// TwinCAT 3 PLC project Test
// ProgramVersion: 3.1.4026.20
// libraries:
//   AUT_Utilities, * (AU-tomation)
//   Tc2_Standard, * (Beckhoff Automation GmbH)
//   Tc2_System, * (Beckhoff Automation GmbH)
//   Tc2_Utilities, * (Beckhoff Automation GmbH)
//   TcUnit, * (www.tcunit.org)
// project tree:
//   / PlcTask.TcTTO
//   POUs/ PRG_TEST.TcPOU, StringBuilder_Test.TcPOU
// real-time tasks:
//   TASK PlcTask: cycle T#10ms, priority 20, ADS port 350

CONFIGURATION Test
    RESOURCE PLC ON TwinCAT3
        TASK PlcTask(INTERVAL := T#10ms, PRIORITY := 20);
        PROGRAM PRG_TEST WITH PlcTask : PRG_TEST;
    END_RESOURCE
END_CONFIGURATION

// ---- POUs/PRG_TEST.TcPOU
{attribute 'no-analysis'}       // Disable SA for entire POU
PROGRAM PRG_TEST
VAR
    {attribute 'analysis' := '-33'}      // Disable SA0033: Unused variable
    _StringBuilder_Test : StringBuilder_Test;
END_VAR

//TcUnit.RUN();
TcUnit.RUN_IN_SEQUENCE();

END_PROGRAM

// ---- POUs/StringBuilder_Test.TcPOU
{attribute 'no-analysis'}       // Disable SA for entire POU
FUNCTION_BLOCK StringBuilder_Test EXTENDS TcUnit.FB_TestSuite

ToStringWithoutAppendEqualsEmptyString();
AppendABCTo123EqualsABC123();
AppendWithFormat();
LeftOfABC123With3EqualsABC();
RightOfABC123With3Equals123();
InsertXYZAt3IntoABC123EqualsABCXYZ123();
MultipleOperations();
RemoveDelimitedSubstring();
AssignDelimitedSubstring();

METHOD AppendABCTo123EqualsABC123
VAR
    {attribute 'analysis' := '-167'}      // Disable SA0167: Temporary FunctionBlock instance
    _StringBuilder : StringBuilder;
    _ResultString : STRING(2048) := '';
    _ExpectedResultString : STRING(2048) := 'ABC123';
END_VAR
TEST('AppendABCTo123EqualsABC123');

_ResultString := _StringBuilder.Append('ABC')
                               .Append('123')
                               .ToString();
                               
AssertEquals_String(Expected := _ExpectedResultString,
             Actual := _ResultString,
             Message := 'The result is not correct');

TEST_FINISHED();
END_METHOD

METHOD AppendWithFormat
VAR
    {attribute 'analysis' := '-167'}      // Disable SA0167: Temporary FunctionBlock instance
    _StringBuilder : StringBuilder;
    _ResultString : STRING(2048) := '';
END_VAR
VAR
    _DIntValue : DINT := 255;
END_VAR
TEST('AppendWithFormat');

// Format DINT variable to hex
_ResultString := _StringBuilder.Reset()
                               .AppendWithFormat(_DIntValue, '%X')
                               .ToString();
                               
AssertEquals_String(Expected := 'FF',
             Actual := _ResultString,
             Message := 'The result is not correct');

// Format DINT variable to 5 digits with leading zeros
_ResultString := _StringBuilder.Reset()
                               .AppendWithFormat(_DIntValue, '%05d')
                               .ToString();
                               
AssertEquals_String(Expected := '  255',
             Actual := _ResultString,
             Message := 'The result is not correct');

TEST_FINISHED();
END_METHOD

METHOD AssignDelimitedSubstring
VAR
    {attribute 'analysis' := '-167'}      // Disable SA0167: Temporary FunctionBlock instance
    _StringBuilder : StringBuilder;
    _ResultString : STRING(2048) := '';
    _StringToAssignTo : STRING(2048);
END_VAR
TEST('AssignDelimitedSubstring');

// Assign first delimited substring
_ResultString := _StringBuilder.Reset()
                               .Append('^/')
                               .Append('ABC/')
                               .Append('123')
                               .AssignDelimitedSubstringTo('/', 1, ADR(_StringToAssignTo), SIZEOF(_StringToAssignTo))
                               .ToString();
                               
AssertEquals_String(Expected := '^',
             Actual := _StringToAssignTo,
             Message := 'Assign first delimited substring failed');

// Assign mid delimited substring
_ResultString := _StringBuilder.Reset()
                               .Append('^/')
                               .Append('ABC/')
                               .Append('123')
                               .AssignDelimitedSubstringTo('/', 2, ADR(_StringToAssignTo), SIZEOF(_StringToAssignTo))
                               .ToString();
                               
AssertEquals_String(Expected := 'ABC',
             Actual := _StringToAssignTo,
             Message := 'Assign mid delimited substring failed');

// Assign last delimited substring
_ResultString := _StringBuilder.Reset()
                               .Append('^/')
                               .Append('ABC/')
                               .Append('123')
                               .AssignDelimitedSubstringTo('/', 3, ADR(_StringToAssignTo), SIZEOF(_StringToAssignTo))
                               .ToString();
                               
AssertEquals_String(Expected := '123',
             Actual := _StringToAssignTo,
             Message := 'Assign last delimited substring failed');

// Assign delimited substring with index 0 (not allowed: return empty string)
_ResultString := _StringBuilder.Reset()
                               .Append('^/')
                               .Append('ABC/')
                               .Append('123')
                               .AssignDelimitedSubstringTo('/', 0, ADR(_StringToAssignTo), SIZEOF(_StringToAssignTo))
                               .ToString();
                               
AssertEquals_String(Expected := '',
             Actual := _StringToAssignTo,
             Message := 'Assign delimited substring with index 0 failed');

// Assign delimited substring with index greater than available (return empty string)
_ResultString := _StringBuilder.Reset()
                               .Append('^/')
                               .Append('ABC/')
                               .Append('123')
                               .AssignDelimitedSubstringTo('/', 4, ADR(_StringToAssignTo), SIZEOF(_StringToAssignTo))
                               .ToString();
                               
AssertEquals_String(Expected := '',
             Actual := _StringToAssignTo,
             Message := 'Assign delimited substring with index greater than available failed');

// Assign delimited substring when only one substring with no delimiters
_ResultString := _StringBuilder.Reset()
                               .Append('ABC')
                               .AssignDelimitedSubstringTo('/', 1, ADR(_StringToAssignTo), SIZEOF(_StringToAssignTo))
                               .ToString();
                               
AssertEquals_String(Expected := 'ABC',
             Actual := _StringToAssignTo,
             Message := 'Assign delimited substring when only one substring with no delimiters');

TEST_FINISHED();
END_METHOD

METHOD InsertXYZAt3IntoABC123EqualsABCXYZ123
VAR
    {attribute 'analysis' := '-167'}      // Disable SA0167: Temporary FunctionBlock instance
    _StringBuilder : StringBuilder;
    _ResultString : STRING(2048) := '';
    _ExpectedResultString : STRING(2048) := 'ABCXYZ123';
END_VAR
TEST('InsertXYZAt3IntoABC123EqualsABCXYZ123');

_ResultString := _StringBuilder.Append('ABC123')
                               .InsertAt('XYZ', 3) 
                               .ToString();
                               
AssertEquals_String(Expected := _ExpectedResultString,
             Actual := _ResultString,
             Message := 'The result is not correct');

TEST_FINISHED();
END_METHOD

METHOD LeftOfABC123With3EqualsABC
VAR
    {attribute 'analysis' := '-167'}      // Disable SA0167: Temporary FunctionBlock instance
    _StringBuilder : StringBuilder;
    _ResultString : STRING(2048) := '';
    _ExpectedResultString : STRING(2048) := 'ABC';
END_VAR
TEST('LeftOfABC123With3EqualsABC');

_ResultString := _StringBuilder.Append('ABC')
                               .Append('123')
                               .Left(3)
                               .ToString();
                               
AssertEquals_String(Expected := _ExpectedResultString,
             Actual := _ResultString,
             Message := 'The result is not correct');

TEST_FINISHED();
END_METHOD

METHOD MultipleOperations
VAR
    {attribute 'analysis' := '-167'}      // Disable SA0167: Temporary FunctionBlock instance
    _StringBuilder : StringBuilder;
    _ResultString : STRING(2048) := '';
END_VAR
TEST('MultipleOperations');

// --- Append ---
_ResultString := _StringBuilder.Reset()
                               .Append('ABC')
                               .Append('123')
                               .ToString();
AssertEquals_STRING('ABC123', _ResultString, 'Append ABC + 123 should produce ABC123');

// --- InsertAt ---
_ResultString := _StringBuilder.Reset()
                               .Append('ABC')
                               .InsertAt('XYZ', 2) // A B C → A B XYZ C
                               .ToString();
AssertEquals_STRING('ABXYZC', _ResultString, 'Insert XYZ at pos 2 should produce ABXYZC');

// --- Left ---
_ResultString := _StringBuilder.Reset()
                               .Append('HELLOWORLD')
                               .Left(5)
                               .ToString();
AssertEquals_STRING('HELLO', _ResultString, 'Left(5) should return HELLO');

// --- Right ---
_ResultString := _StringBuilder.Reset()
                               .Append('HELLOWORLD')
                               .Right(5)
                               .ToString();
AssertEquals_STRING('WORLD', _ResultString, 'Right(5) should return WORLD');

// --- RemoveAt ---
_ResultString := _StringBuilder.Reset()
                               .Append('ABCDE')
                               .RemoveAt(2, 2) // remove BC → ADE
                               .ToString();
AssertEquals_STRING('ADE', _ResultString, 'RemoveAt(2,2) should remove BC and produce ADE');

// --- Reset ---
_ResultString := _StringBuilder.Reset()
                               .ToString();
AssertEquals_STRING('', _ResultString, 'Reset should produce empty string');

TEST_FINISHED();
END_METHOD

METHOD RemoveDelimitedSubstring
VAR
    {attribute 'analysis' := '-167'}      // Disable SA0167: Temporary FunctionBlock instance
    _StringBuilder : StringBuilder;
    _ResultString : STRING(2048) := '';
END_VAR
TEST('RemoveDelimitedSubstring');

// Remove first delimited substring
_ResultString := _StringBuilder.Reset()
                               .Append('^/')
                               .Append('ABC/')
                               .Append('123')
                               .RemoveDelimitedSubstring('/', 1)
                               .ToString();
                               
AssertEquals_String(Expected := 'ABC/123',
             Actual := _ResultString,
             Message := 'Remove first delimited substring failed');

// Remove mid delimited substring
_ResultString := _StringBuilder.Reset()
                               .Append('^/')
                               .Append('ABC/')
                               .Append('123')
                               .RemoveDelimitedSubstring('/', 2)
                               .ToString();
                               
AssertEquals_String(Expected := '^/123',
             Actual := _ResultString,
             Message := 'Remove mid delimited substring failed');

// Remove last delimited substring
_ResultString := _StringBuilder.Reset()
                               .Append('^/')
                               .Append('ABC/')
                               .Append('123')
                               .RemoveDelimitedSubstring('/', 3)
                               .ToString();
                               
AssertEquals_String(Expected := '^/ABC',
             Actual := _ResultString,
             Message := 'Remove last delimited substring failed');

// Remove delimited substring with index 0 (not allowed: no operations)
_ResultString := _StringBuilder.Reset()
                               .Append('^/')
                               .Append('ABC/')
                               .Append('123')
                               .RemoveDelimitedSubstring('/', 0)
                               .ToString();
                               
AssertEquals_String(Expected := '^/ABC/123',
             Actual := _ResultString,
             Message := 'Remove delimited substring with index 0 failed');

// Remove delimited substring with index greater than available (no operations)
_ResultString := _StringBuilder.Reset()
                               .Append('^/')
                               .Append('ABC/')
                               .Append('123')
                               .RemoveDelimitedSubstring('/', 4)
                               .ToString();
                               
AssertEquals_String(Expected := '^/ABC/123',
             Actual := _ResultString,
             Message := 'Remove delimited substring with index greater than available failed');

// Remove delimited substring when only one substring with no delimiters
_ResultString := _StringBuilder.Reset()
                               .Append('ABC')
                               .RemoveDelimitedSubstring('/', 1)
                               .ToString();
                               
AssertEquals_String(Expected := '',
             Actual := _ResultString,
             Message := 'Remove delimited substring when only one substring with no delimiters');

TEST_FINISHED();
END_METHOD

METHOD RightOfABC123With3Equals123
VAR
    {attribute 'analysis' := '-167'}      // Disable SA0167: Temporary FunctionBlock instance
    _StringBuilder : StringBuilder;
    _ResultString : STRING(2048) := '';
    _ExpectedResultString : STRING(2048) := '123';
END_VAR
TEST('RightOfABC123With3Equals123');

_ResultString := _StringBuilder.Append('ABC')
                               .Append('123')
                               .Right(3)
                               .ToString();
                               
AssertEquals_String(Expected := _ExpectedResultString,
             Actual := _ResultString,
             Message := 'The result is not correct');

TEST_FINISHED();
END_METHOD

METHOD ToStringWithoutAppendEqualsEmptyString
VAR
    {attribute 'analysis' := '-167'}      // Disable SA0167: Temporary FunctionBlock instance
    _StringBuilder : StringBuilder;
    _ResultString : STRING(2048) := '';
    _ExpectedResultString : STRING(2048) := '';
END_VAR
TEST('ToStringWithoutAppendEqualsEmptyString');

_ResultString := _StringBuilder.ToString();
                               
AssertEquals_String(Expected := _ExpectedResultString,
             Actual := _ResultString,
             Message := 'The result is not correct');

TEST_FINISHED();
END_METHOD

END_FUNCTION_BLOCK
